PROGRAM MAIN
VAR
	Apotentiometer AT %I*: INT := 0;
	Npotentiometer AT %I*: INT;
	NScale AT %I*: INT := 100;
END_VAR

Apotentiometer := LREAL_TO_INT (F_Scale(Npotentiometer, 0,32767,0,NScale));

END_PROGRAM

(* stored: Version 1.1.0.1, ProductVersion 3.1.4024.12
   POU MAIN: Id {9ab3aa86-362b-495d-b39a-3a88b0b7b42b}, SpecialFunc None *)
